FUNCTION_BLOCK Aux_IX (* Input service interface function block for boolean input data *)
  (* Description: Copyright (c) 2014, 2015 fortiss GmbH This program and the accompanying materials are made available under the terms of the Eclipse Public License 2.0 which is available at https://www.eclipse.org/legal/epl-2.0/ SPDX-License-Identifier: EPL-2.0 *)
  (* Version 1.0, 2014-08-26, Waldemar Eisenmenger, fortiss GmbH *)
  (* Version 1.1, 2014-08-30, Alois Zoitl, fortiss GmbH *)
  (* Version 1.2, 2015-06-10, Monika Wenger, fortiss GmbH *)
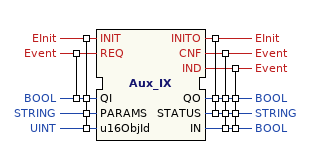
  EVENT_INPUT
    INIT : EInit WITH QI, PARAMS, u16ObjId; (* Service Initialization *)
    REQ WITH QI; (* Service Request *)
  END_EVENT
  EVENT_OUTPUT
    INITO : EInit WITH QO, STATUS; (* Initialization Confirm *)
    CNF WITH QO, STATUS, IN; (* Confirmation of Requested Service *)
    IND WITH QO, STATUS, IN; (* Indication from Resource *)
  END_EVENT
  VAR_INPUT
    QI : BOOL; (* Event Input Qualifier *)
    PARAMS : STRING; (* Service Parameters *)
    u16ObjId : UINT := isobus::ID_NULL; (* Object ID *)
  END_VAR
  VAR_OUTPUT
    QO : BOOL; (* Event Output Qualifier *)
    STATUS : STRING; (* Service Status *)
    IN : BOOL; (* Input data from resource *)
  END_VAR
END_FUNCTION_BLOCK
